# EPICS IOC start-up script: iocsh/evr-pcie-300dc-init.iocsh
#- ###   ESS PCIE EVR 300DC Configuration iocsh     ###
#- ####################################################
#- >> Mandatory
#- PCIID          - PCI Address
#- S              - System name for Record
#- DEV            - Device Name for EVR and for Record name
#-                  In DB, (SYS)-$(D):Signal-SD
#-                  In iocsh, (S)-$(DEV):Signal-SD
#- >> Optional
#- EVTCLOCKRATE   - Event Clock Rate, ESS 88.0525
#  RT             - software timestamp source w/o RT thread scheduling
#                   wtRT : diable software timestamp source
#                   woRT : Default, enable it.
#- ####################################################
#-iocshLoad("$(mrfioc2_DIR)/evr-pcie-300dc.iocsh", "S=$(IOC), DEV=$(DEV), PCIID=03:00.0")
#-iocshLoad("$(mrfioc2_DIR)/evr-pcie-300dc.iocsh", "S=$(IOC), DEV=$(DEV), PCIID=03:00.0, RT=wtRT")
#-
mrmEvrSetupPCI("$(DEV)",  "$(PCIID)")
dbLoadRecords("evr-pcie-300dc-ess.db","EVR=$(DEV), SYS=$(S), D=$(DEV), FEVT=$(EVTCLOCKRATE=88.0525)")
iocshRun('$(SWTIMESTAMP_$(RT=woRT)=) var(evrMrmTimeNSOverflowThreshold, 1000000)', "SWTIMESTAMP_wtRT=#")
#-
#- Don't forget the new line
